Staubli VAL3: onF7Event.pgx

program onF7Event(string x_sName)
  local num l_nMax
begin
  // look if the bButton is enable
  if bButton[6]
    // BACK
    call pallet:back(x_sName)
    // refresh it
    call buildList()
    use:bUseRefresh=true
  endIf
end
